FUNCTION_BLOCK ASSEMBLE_AB_FROM_AQ (* this Function combines the 4 AQ (QUARTER) adapters to a AB (BYTE) *)
  (* Standard: 61499-2; Description: Copyright (c) 2026 Meisterschulen am Ostbahnhof SPDX-License-Identifier: EPL-2.0 *)
  (* Version 1.0, 2026-05-16, Franz Höpfinger, Meisterschulen am Ostbahnhof, initial API and implementation and/or initial documentation *)
  PACKAGE adapter::assembling;
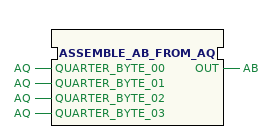
  SOCKETS
    QUARTER_BYTE_00 : adapter::types::unidirectional::AQ; (* Quarter 0 *)
    QUARTER_BYTE_01 : adapter::types::unidirectional::AQ; (* Quarter 1 *)
    QUARTER_BYTE_02 : adapter::types::unidirectional::AQ; (* Quarter 2 *)
    QUARTER_BYTE_03 : adapter::types::unidirectional::AQ; (* Quarter 3 *)
  END_SOCKETS
  PLUGS
    OUT : adapter::types::unidirectional::AB; (* BYTE Output *)
  END_PLUGS
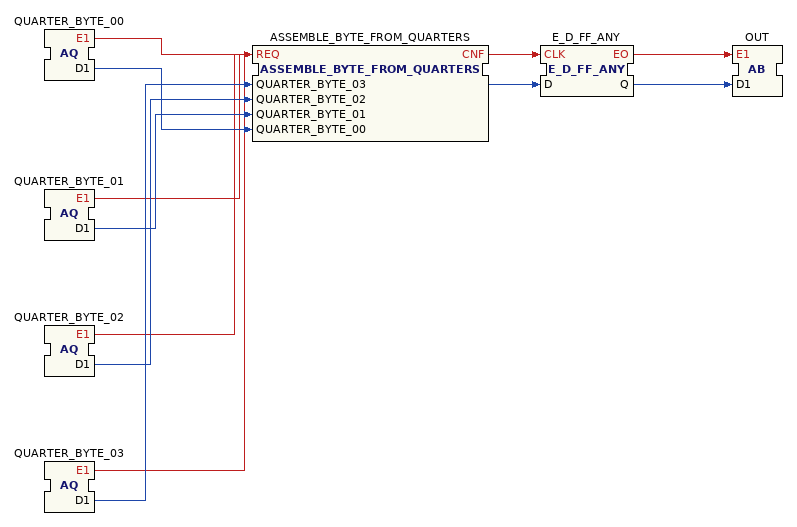
  FBS
    ASSEMBLE_BYTE_FROM_QUARTERS : eclipse4diac::utils::assembling::ASSEMBLE_BYTE_FROM_QUARTERS;
    E_D_FF_ANY : iec61499::events::E_D_FF_ANY;
  END_FBS
  EVENT_CONNECTIONS
    QUARTER_BYTE_00.E1 TO ASSEMBLE_BYTE_FROM_QUARTERS.REQ;
    QUARTER_BYTE_01.E1 TO ASSEMBLE_BYTE_FROM_QUARTERS.REQ;
    QUARTER_BYTE_02.E1 TO ASSEMBLE_BYTE_FROM_QUARTERS.REQ;
    QUARTER_BYTE_03.E1 TO ASSEMBLE_BYTE_FROM_QUARTERS.REQ;
    ASSEMBLE_BYTE_FROM_QUARTERS.CNF TO E_D_FF_ANY.CLK;
    E_D_FF_ANY.EO TO OUT.E1;
  END_CONNECTIONS
  DATA_CONNECTIONS
    ASSEMBLE_BYTE_FROM_QUARTERS. TO E_D_FF_ANY.D;
    E_D_FF_ANY.Q TO OUT.D1;
    QUARTER_BYTE_03.D1 TO ASSEMBLE_BYTE_FROM_QUARTERS.QUARTER_BYTE_03;
    QUARTER_BYTE_02.D1 TO ASSEMBLE_BYTE_FROM_QUARTERS.QUARTER_BYTE_02;
    QUARTER_BYTE_01.D1 TO ASSEMBLE_BYTE_FROM_QUARTERS.QUARTER_BYTE_01;
    QUARTER_BYTE_00.D1 TO ASSEMBLE_BYTE_FROM_QUARTERS.QUARTER_BYTE_00;
  END_CONNECTIONS
END_FUNCTION_BLOCK
